# EPICS autosave request: iocBoot/ioc13bmc_linux/Galil_positions.req
file "CARS_32_motor_positions.req",     P=$(P)
file "CARS_8_motor_positions_sub.req",  P=$(P), M1=m47, M2=m48, M3=m49, M4=m50, M5=m51, M6=m52, M7=m53, M8=m54
file "CARS_8_motor_positions_sub.req",  P=$(P), M1=m63, M2=m64, M3=m65, M4=m66, M5=m67, M6=m68, M7=m69, M8=m70
file "CARS_8_motor_positions_sub.req",  P=$(P), M1=m71, M2=m72, M3=m73, M4=m74, M5=m75, M6=m76, M7=m77, M8=m78
